INTERFACE ITF_TaskObserver EXTENDS __System.IQueryInterface

PROPERTY activity : E_SocketCommStateMachine
GET
END_GET
SET
END_SET
END_PROPERTY

PROPERTY complete : BOOL
GET
END_GET
SET
END_SET
END_PROPERTY

PROPERTY error : BOOL
GET
END_GET
SET
END_SET
END_PROPERTY

PROPERTY error_id : UDINT
GET
END_GET
SET
END_SET
END_PROPERTY

END_INTERFACE

(* stored: Version 1.1.0.1, ProductVersion 3.1.4024.15
   Itf ITF_TaskObserver: Id {85e3cb91-aef8-4900-81d3-52daa497447f}
   Property activity: Id {b5a0bc98-62f1-40d7-973d-e53181ef602a}
   Get Get: Id {3ffb790a-601d-447f-a52d-7d51f645bc6f}
   Set Set: Id {015aced3-2151-4648-9cce-f21ea1d3f351}
   Property complete: Id {89d65bc5-48c5-41d8-a00c-d66c493312e4}
   Get Get: Id {6a748588-3fc8-4468-8b76-3852701abb15}
   Set Set: Id {44298304-d244-4a8c-b9a3-c4f8415e6705}
   Property error: Id {60f8f907-3200-490c-b186-fb182d4db388}
   Get Get: Id {087d9acd-fa7b-4835-8723-8d1cd48b8a97}
   Set Set: Id {ac37d9e0-bb05-496f-8a64-50ae375ec752}
   Property error_id: Id {de092223-029b-494c-85ec-3d21c7127063}
   Get Get: Id {6adb83be-7cda-4f05-8067-324d278fea6e}
   Set Set: Id {8861e922-0d4f-4bef-9d86-e2f8239957c4} *)
